Fanuc KAREL source: kt00621.KL

PROGRAM KT00621
%NOLOCKGROUP
VAR
B1:BOOLEAN;B2:BOOLEAN;OUT:BOOLEAN
BEGIN
--
--
B1=TRUE
B2=FALSE
B1=TRUE
B2=FALSE
OUT=B1
END KT00621
